{attribute addProperty BoxType "EK1122-0000-0018"}
{attribute addProperty Id "Beckhoff_APS1xxxsub_EK1100EK1100_179A0949162A_0001_APS1003_7000_0016APS1003_D64416202098262.25"}
{attribute addProperty CRC "2246513059"}
{attribute addProperty SizeInBites "2114"}
{attribute addProperty SizeInBytes "264.25"}
TYPE Beckhoff_APS1xxxEK1122_85E711A3 EXTENDS EK1122_179A0949 :
STRUCT
	{attribute addProperty Name "Beckhoff_APS1xxxsub_EK1100"}
	Beckhoff_APS1xxxsub_EK1100 : EK1100_179A0949;
	{attribute addProperty Name "A_0001_APS1003_7000_0016"}
	A_0001_APS1003_7000_0016 : APS1003_D6441620;
END_STRUCT
END_TYPE

(* stored: Version 1.2.0.0, ProductVersion 3.1.4024.9
   DUT Beckhoff_APS1xxxEK1122_85E711A3: Id {71ea8052-e750-4fbe-8a18-de30f464bbad} *)
